// Block: Decoiler2_PERS

DATA_BLOCK Decoiler2_PERS
VERSION : 0.1
   NON_RETAIN
   VAR
      PersistentValues : Decoiler_Pers;
   END_VAR

BEGIN
   // No initialization required
END_DATA_BLOCK
